PROGRAM POU_DIVIDE
VAR
	Result:REAL;
	Value01:REAL;
	Value02:REAL;
END_VAR

IF MAIN.Value02=0 THEN
	;
	ELSE
		Result:=MAIN.Value01/MAIN.Value02;
END_IF

END_PROGRAM

(* stored: Version 1.1.0.1, ProductVersion 3.1.4024.4
   POU POU_DIVIDE: Id {fb69de74-b83b-4c3c-98d4-e8185c7723da}, SpecialFunc None *)
